INTERFACE PUBLIC ClearingCommands

METHOD PUBLIC Abort
END_METHOD

METHOD PUBLIC StateComplete
END_METHOD

END_INTERFACE

(* stored: Version 1.1.0.1, ProductVersion 3.1.4026.12
   Itf ClearingCommands: Id {e5c1cdf7-471e-0292-28be-8a8a5b1d0479}
   Method Abort: Id {f9aa4c48-18d5-4b8f-9204-1a96d7f5145c}
   Method StateComplete: Id {520dd82a-14d0-4ae5-b79a-a7ce2ba113f7} *)
